# EPICS autosave request: ADCore/ADApp/Db/NDFileJPEG_settings.req
$(P)$(R)JPEGQuality
